(* CODESYS project FaultReset.xml

Project tree, tasks and I/O mapping:
  function block FaultReset [LD]
*)

// FaultReset
FUNCTION_BLOCK FaultReset
VAR_INPUT
END_VAR
VAR_OUTPUT
	IceMaker: BOOL;
	
END_VAR
VAR
END_VAR

// NETWORK 1

END_FUNCTION_BLOCK
